TYPE DUT_MB :
STRUCT
	
	bExecute	:BOOL;	
	bBusy		:BOOL;
	bError		:BOOL;
	nErrId		:UDINT;
	
END_STRUCT
END_TYPE

(* stored: Version 1.1.0.1, ProductVersion 3.1.4024.6
   DUT DUT_MB: Id {c3253826-c977-4f56-a3e6-d47d86bf0ac6} *)
